FUNCTION_BLOCK CornerHarris (* openCV CornerHarris *)
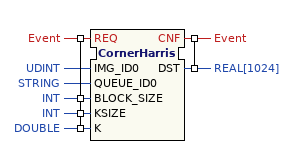
  EVENT_INPUT
    REQ WITH IMG_ID, QUEUE_ID, BLOCK_SIZE, KSIZE, K;
  END_EVENT
  EVENT_OUTPUT
    CNF WITH DST;
  END_EVENT
  VAR_INPUT
    IMG_ID0 : UDINT;
    QUEUE_ID0 : STRING;
    BLOCK_SIZE : INT;
    KSIZE : INT;
    K : DOUBLE;
  END_VAR
  VAR_OUTPUT
    DST : ARRAY [0..1023] OF REAL;
  END_VAR
END_FUNCTION_BLOCK
